{attribute 'pack_mode' := '1'}
TYPE ST_1100_Position_initialization_started EXTENDS ST_SupervisorHeader :
STRUCT
END_STRUCT
END_TYPE

(* stored: Version 1.1.0.1, ProductVersion 3.1.4026.17
   DUT ST_1100_Position_initialization_started: Id {da62d4de-c1a5-46c7-a24c-b038a481be71} *)
